(* PLC project PRG_00_ACQUISITION_CFC.project, Dragage CODESYS CODESYS V3.5 SP19 Patch 1 *)
(* stored: creationDateTime 2026-08-01T00:00:00, modificationDateTime 2026-08-01T00:00:00 *)

PROGRAM PRG_00_ACQUISITION_CFC
  VAR
    instJoystick : FB_Joystick;
    instEncoderAbsM1 : FB_Encoder_Abs;
    instEncoderScaleM1 : FB_Encoder_Scale;
    instHomingM1 : FB_Encoder_Homing;
    instEncoderAbsM2 : FB_Encoder_Abs;
    instEncoderScaleM2 : FB_Encoder_Scale;
    instHomingM2 : FB_Encoder_Homing;
    instPosDecoderM3 : FB_Translation_PositionDecoder;
  END_VAR

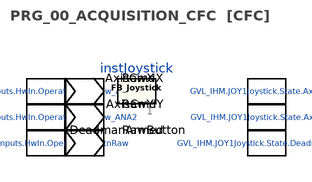
(* CFC diagram, written out as Structured Text *)
instJoystick(RawX := PRG_00_Inputs.HwIn.Operator.JoyXRaw_ANA1, RawY := PRG_00_Inputs.HwIn.Operator.JoyYRaw_ANA2, RawButton := PRG_00_Inputs.HwIn.Operator.JoyBtnRaw);
GVL_IHM.JOY1Joystick.State.AxisCmdX := instJoystick.AxisCmdX;
GVL_IHM.JOY1Joystick.State.AxisCmdY := instJoystick.AxisCmdY;
GVL_IHM.JOY1Joystick.State.DeadmanArmed := instJoystick.DeadmanArmed;
END_PROGRAM
